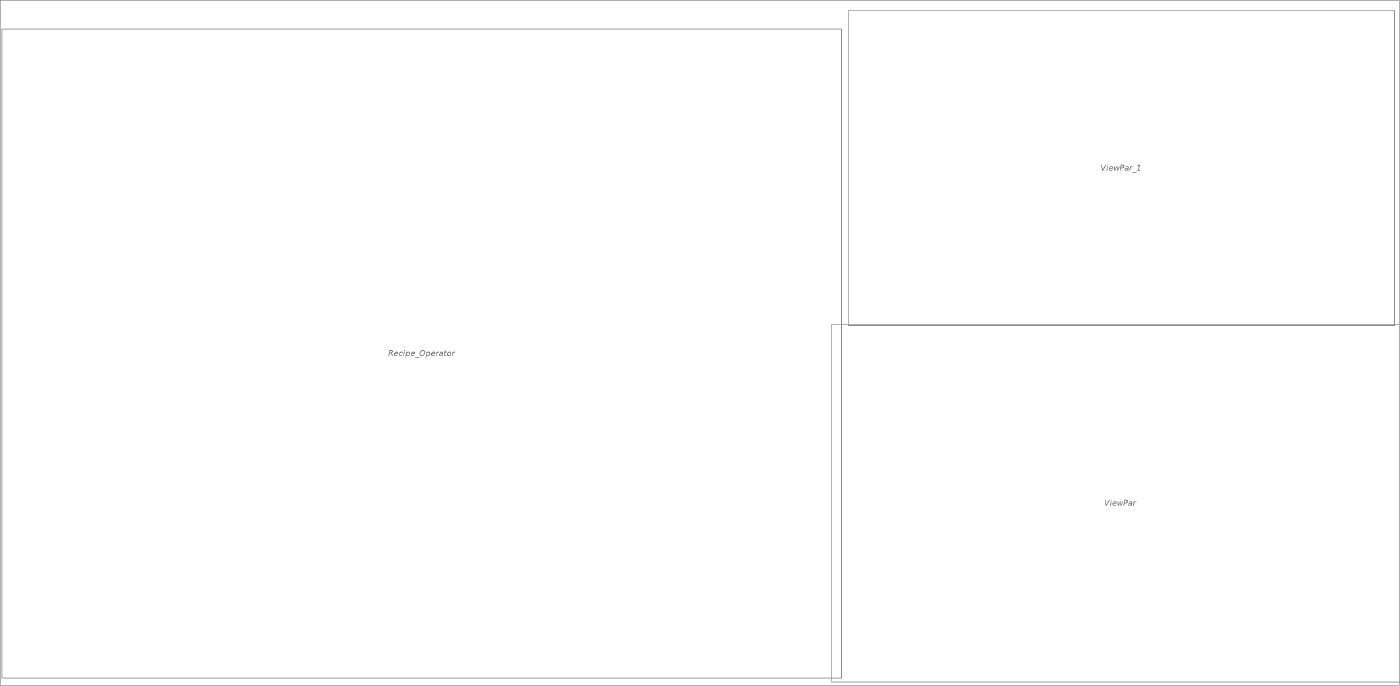
VISUALIZATION Operator  // 1755x860
    Frame (1042,406 724x449)
        shows ViewPar()
    Frame (2,36 1053x814)
        shows Recipe_Operator()
    Frame (1063,13 685x395)
        shows ViewPar_1()
END_VISUALIZATION

(* stored: Version 1.1.0.1, ProductVersion 3.1.4024.12
   Visu Operator: Id {a7bace33-8ef3-4b7c-8c1a-d70652735a5b} *)
